FUNCTION Init_PB_Mom_250x75 : INT

VAR_INPUT
END_VAR

VAR

END_VAR

VAR_IN_OUT
	COMP:TS_Component;
END_VAR

COMP.B_TYPE:=0;
COMP.size:=3;

END_FUNCTION

(* stored: Version 1.1.0.1, ProductVersion 3.1.4020.12
   POU Init_PB_Mom_250x75: Id {2b9ef975-c776-4f5b-84b3-24bcb9df45c8}, SpecialFunc None *)
